// SIMATIC S7-200 project (STEP 7-Micro/WIN), CPU 221 REL 01.10

ORGANIZATION_BLOCK MAIN:OB1
TITLE=PROGRAM COMMENTS
BEGIN
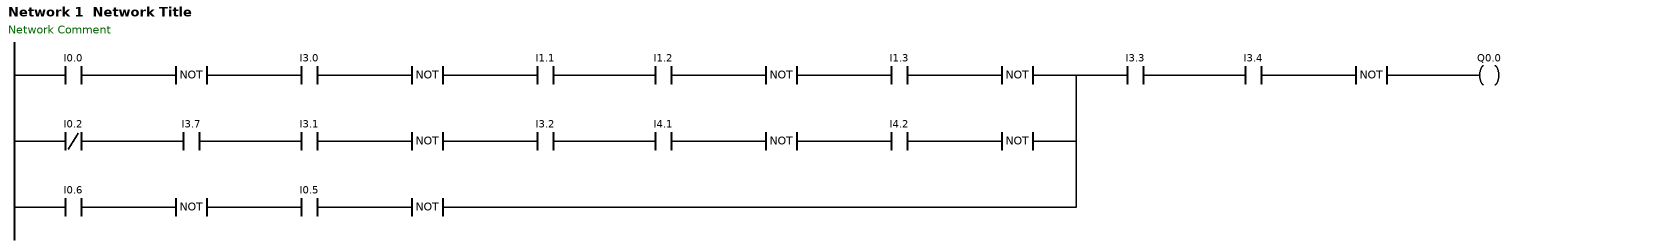
Network 1 // Network Title
// Network Comment
LD     I0.0
NOT
A      I3.0
NOT
A      I1.1
A      I1.2
NOT
A      I1.3
NOT
LDN    I0.2
A      I3.7
A      I3.1
NOT
A      I3.2
A      I4.1
NOT
A      I4.2
NOT
OLD
LD     I0.6
NOT
A      I0.5
NOT
OLD
A      I3.3
A      I3.4
NOT
=      Q0.0
END_ORGANIZATION_BLOCK
